RoboDK station: nameHW.rdk

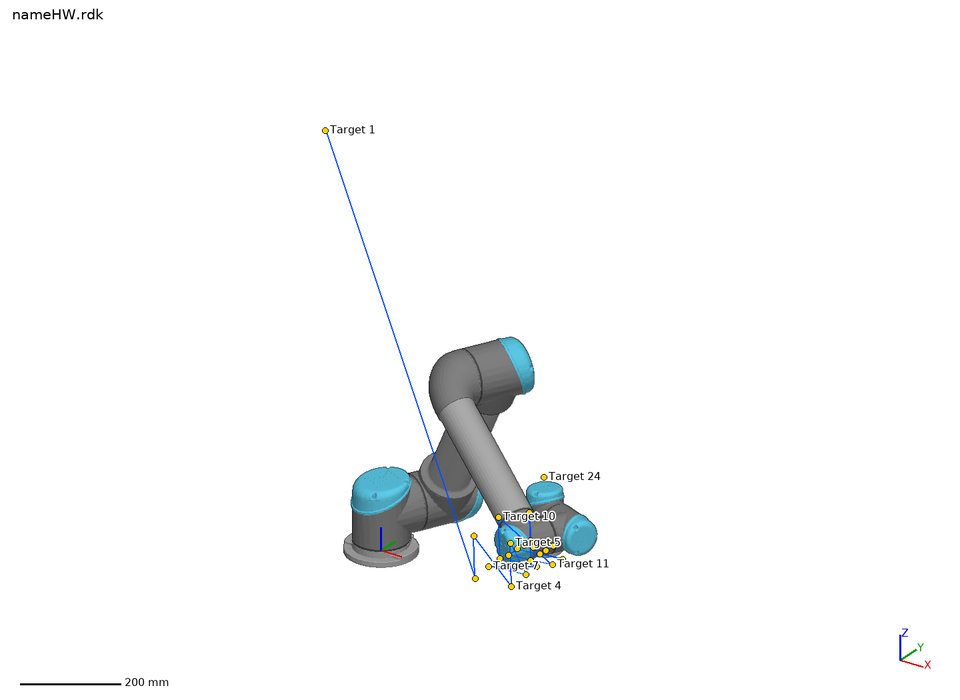
[picture v0: the station drawn from its stored meshes, robots at their saved joint values, targets as dots, program paths as lines]
Station nameHW (saved by RoboDK 5.4.1). Poses are relative to the parent item; angles as X-Y-Z fixed-axis rotations.
  - frame UR5 Base at (0, 0, 0) mm
    - robot UR5: 6 axes, payload 5 kg, reach 850 mm, repeatability 0.1 mm, weight 18.4 kg
        modified DH rows (alpha deg, a mm, theta deg, d mm): 0, 0, 0, 89.2; 90, 0, 180, 0; 0, 425, 0, 0; 0, 392.43, 0, 109; -90, 0, 0, 93.65; 90, 0, 180, 82
        joint limits [-360, -360, -360, -360, -360, -360] to [360, 360, 360, 360, 360, 360]; home [0, -90, -90, 0, 90, 0]; saved at [154.945, -59.412, 90.192, 56.995, 89.781, -29.068]
    - target Target 7 (Cartesian target) at (413.27, -220.03, 168.94) mm, rotated rx 177.95 ry 0.89 rz 94 deg; joints [138.353, -60.309, 91.655, 56.584, 89.155, -45.649] of UR5
    - target Target 8 (Cartesian target) at (494.97, -170.3, 171.3) mm, rotated rx 177.95 ry 0.89 rz 94 deg; joints [148.922, -53.776, 80.298, 61.288, 89.549, -35.087] of UR5
    - target Target 9 (Cartesian target) at (410.34, -176.27, 168.26) mm, rotated rx 177.95 ry 0.89 rz 94 deg; joints [142.495, -62.815, 95.789, 54.901, 89.306, -41.51] of UR5
    - target Target 6 (Cartesian target) at (499.82, -213.93, 172.05) mm, rotated rx 177.95 ry 0.89 rz 94 deg; joints [145.172, -51.245, 75.806, 63.283, 89.406, -38.834] of UR5
    - target Target 5 (Cartesian target) at (500.39, -268.72, 263.98) mm, rotated rx 177.95 ry 0.89 rz 94 deg; joints [140.586, -51.868, 62.76, 77.007, 89.236, -43.417] of UR5
    - target Target 4 (Cartesian target) at (503.88, -269.95, 169.1) mm, rotated rx 177.95 ry 0.89 rz 94 deg; joints [140.716, -47.371, 69.437, 65.831, 89.241, -43.287] of UR5
    - target Target 3 (Cartesian target) at (416.54, -274.68, 258.01) mm, rotated rx 177.95 ry 0.89 rz 94 deg; joints [133.81, -61.405, 79.08, 70.328, 88.993, -50.19] of UR5
    - target Target 2 (Cartesian target) at (419.93, -275.87, 166.08) mm, rotated rx 177.95 ry 0.89 rz 94 deg; joints [134, -56, 85, 59, 89, -50] of UR5
    - target Target 1 (joint target) at (0, -191, 1000.28) mm, rotated rx -90 ry 0 rz 180 deg; joints [0, -90, 0, -90, 0, 0] of UR5
    - target Target 10 (Cartesian target) at (407.08, -175.12, 256.68) mm, rotated rx 177.95 ry 0.89 rz 94 deg; joints [142.351, -68.696, 90.077, 66.495, 89.301, -41.654] of UR5
    - target Target 11 (Cartesian target) at (513.09, -142.12, 168.88) mm, rotated rx 177.95 ry 0.89 rz 94 deg; joints [152.655, -52.503, 78.491, 61.798, 89.692, -31.356] of UR5
    - target Target 12 (Cartesian target) at (412.36, -149.23, 165.26) mm, rotated rx 177.95 ry 0.89 rz 94 deg; joints [145.602, -63.539, 97.451, 53.927, 89.423, -38.405] of UR5
    - target Target 13 (Cartesian target) at (410, -115.43, 164.74) mm, rotated rx 177.95 ry 0.89 rz 94 deg; joints [149.363, -64.968, 99.779, 52.996, 89.565, -34.646] of UR5
    - target Target 14 (Cartesian target) at (513.7, -108.11, 168.46) mm, rotated rx 177.95 ry 0.89 rz 94 deg; joints [156.103, -53.414, 80.129, 61.056, 89.826, -27.911] of UR5
    - target Target 15 (Cartesian target) at (461.78, -111.77, 166.6) mm, rotated rx 177.95 ry 0.89 rz 94 deg; joints [153.079, -59.345, 90.436, 56.692, 89.708, -30.933] of UR5
    - target Target 16 (Cartesian target) at (464.24, -146.92, 167.14) mm, rotated rx 177.95 ry 0.89 rz 94 deg; joints [149.429, -57.973, 88.08, 57.699, 89.568, -34.58] of UR5
    - target Target 17 (Cartesian target) at (460.41, -145.57, 271.13) mm, rotated rx 177.95 ry 0.89 rz 94 deg; joints [149.333, -64.124, 81.154, 70.777, 89.564, -34.676] of UR5
    - target Target 18 (Cartesian target) at (412.29, -74.29, 166.4) mm, rotated rx 177.95 ry 0.89 rz 94 deg; joints [154.657, -65.914, 100.938, 52.752, 89.77, -29.356] of UR5
    - target Target 19 (Cartesian target) at (414.03, -99.21, 166.79) mm, rotated rx 177.95 ry 0.89 rz 94 deg; joints [151.622, -65.15, 99.692, 53.249, 89.652, -32.389] of UR5
    - target Target 20 (Cartesian target) at (435.49, -97.69, 167.56) mm, rotated rx 177.95 ry 0.89 rz 94 deg; joints [153.166, -62.807, 95.871, 54.718, 89.712, -30.846] of UR5
    - target Target 21 (Cartesian target) at (433.64, -71.28, 167.15) mm, rotated rx 177.95 ry 0.89 rz 94 deg; joints [156.273, -63.576, 97.159, 54.188, 89.832, -27.742] of UR5
    - target Target 22 (Cartesian target) at (463.79, -69.15, 168.23) mm, rotated rx 177.95 ry 0.89 rz 94 deg; joints [158.061, -60.191, 91.537, 56.42, 89.902, -25.955] of UR5
    - target Target 23 (Cartesian target) at (465.75, -97.05, 168.67) mm, rotated rx 177.95 ry 0.89 rz 94 deg; joints [154.945, -59.412, 90.192, 56.995, 89.781, -29.068] of UR5
    - target Target 24 (Cartesian target) at (459.87, -94.98, 328.2) mm, rotated rx 177.95 ry 0.89 rz 94 deg; joints [154.868, -67.778, 77.885, 77.668, 89.778, -29.145] of UR5
  - program Prog1 (24 instructions, listed below)
  - program Prog2 (2 instructions, listed below)
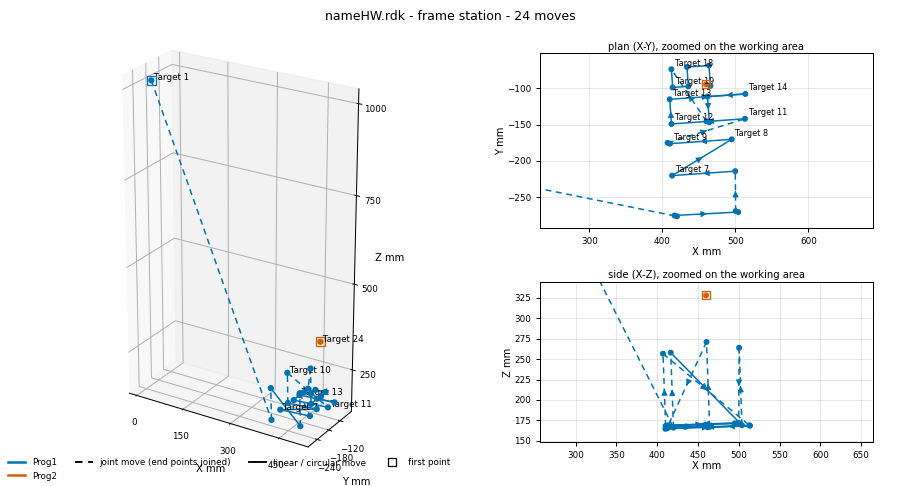
[picture p0: tool path of nameHW.rdk in frame station, 24 of 24 moves have a stored position in this frame; points joined in program order, loops and branches not executed]

--- program Prog1 (robot UR5) ---
  Set Ref.: UR5 Base
  MoveJ (Target 1)
  MoveJ (Target 2) to (419.93, -275.87, 166.08) mm, rotated rx 177.95 ry 0.89 rz 94 deg; joints [134, -56, 85, 59, 89, -50]
  MoveJ (Target 3) to (416.54, -274.68, 258.01) mm, rotated rx 177.95 ry 0.89 rz 94 deg; joints [133.81, -61.405, 79.08, 70.328, 88.993, -50.19]
  MoveL (Target 4) to (503.88, -269.95, 169.1) mm, rotated rx 177.95 ry 0.89 rz 94 deg; joints [140.716, -47.371, 69.437, 65.831, 89.241, -43.287]
  MoveJ (Target 5) to (500.39, -268.72, 263.98) mm, rotated rx 177.95 ry 0.89 rz 94 deg; joints [140.586, -51.868, 62.76, 77.007, 89.236, -43.417]
  MoveJ (Target 6) to (499.82, -213.93, 172.05) mm, rotated rx 177.95 ry 0.89 rz 94 deg; joints [145.172, -51.245, 75.806, 63.283, 89.406, -38.834]
  MoveL (Target 7)
  MoveL (Target 8)
  MoveL (Target 9)
  MoveJ (Target 10)
  MoveJ (Target 11)
  MoveL (Target 12)
  MoveL (Target 13)
  MoveL (Target 14)
  MoveL (Target 15)
  MoveL (Target 16)
  MoveJ (Target 17)
  MoveJ (Target 18)
  MoveL (Target 19)
  MoveL (Target 20)
  MoveL (Target 21)
  MoveL (Target 22)
  MoveL (Target 23)

--- program Prog2 (robot UR5) ---
  Set Ref.: UR5 Base
  MoveJ (Target 24)
